(* IEC 61131-3 sources: JaccoSigma/tempclass/Class/SDM081, 1 file *)

(* ---- SDM081.st ---- *)
(*!
<Class
	Name               = "SDM081"
	Revision           = "1.11"
	RealtimeTask       = "false"
	CyclicTask         = "false"
	BackgroundTask     = "false"
	Sigmatek           = "true"
	OSInterface        = "false"
	HighPriority       = "false"
	Automatic          = "false"
	UpdateMode         = "Prescan"
	IconPath           = ".\Class\sdm.ico"
	SharedCommandTable = "true"
	Objectsize         = "(532,120)">
	<Channels>
		<Server Name="Safe_Input1" Visualized="true" Initialize="false" WriteProtected="true" Retentive="false" Comment="State of input (read only)&#13;&#10;&#13;&#10;-1..Error&#13;&#10; 0..Input Low&#13;&#10; 1..Input High"/>
		<Server Name="Safe_Input2" Visualized="true" Initialize="false" WriteProtected="true" Retentive="false" Comment="State of input (read only)&#13;&#10;&#13;&#10;-1..Error&#13;&#10; 0..Input Low&#13;&#10; 1..Input High"/>
		<Server Name="Safe_Input3" Visualized="true" Initialize="false" WriteProtected="true" Retentive="false" Comment="State of input (read only)&#13;&#10;&#13;&#10;-1..Error&#13;&#10; 0..Input Low&#13;&#10; 1..Input High"/>
		<Server Name="Safe_Input4" Visualized="true" Initialize="false" WriteProtected="true" Retentive="false" Comment="State of input (read only)&#13;&#10;&#13;&#10;-1..Error&#13;&#10; 0..Input Low&#13;&#10; 1..Input High"/>
		<Server Name="Safe_Input5" Visualized="true" Initialize="false" WriteProtected="true" Retentive="false" Comment="State of input (read only)&#13;&#10;&#13;&#10;-1..Error&#13;&#10; 0..Input Low&#13;&#10; 1..Input High"/>
		<Server Name="Safe_Input6" Visualized="true" Initialize="false" WriteProtected="true" Retentive="false" Comment="State of input (read only)&#13;&#10;&#13;&#10;-1..Error&#13;&#10; 0..Input Low&#13;&#10; 1..Input High"/>
		<Server Name="Safe_Output1" Visualized="true" Initialize="false" WriteProtected="true" Retentive="false" Comment="State of output (read only)&#13;&#10;&#13;&#10;-1..Error&#13;&#10; 0..Output Low&#13;&#10; 1..Output High"/>
		<Server Name="Safe_Output2" Visualized="true" Initialize="false" WriteProtected="true" Retentive="false" Comment="State of output (read only)&#13;&#10;&#13;&#10;-1..Error&#13;&#10; 0..Output Low&#13;&#10; 1..Output High"/>
		<Server Name="SafeIOError" Visualized="true" Initialize="false" WriteProtected="true" Retentive="false" Comment="Shows which safe in/outputs are in error.&#13;&#10;The in/outputs are bitcoded.&#13;&#10;Bit0 = Input1&#13;&#10;Bit1 = Input2&#13;&#10;Bit2 = Input3&#13;&#10;Bit3 = Input1&#13;&#10;Bit4 = Input2&#13;&#10;Bit5 = Input3&#13;&#10;Bit6 = Output1&#13;&#10;Bit7 = Output2"/>
		<Server Name="Unsafe_Output1" Visualized="true" Initialize="false" WriteProtected="false" Retentive="false" Comment="State of output (write only; default value: 0)&#13;&#10;&#13;&#10;If safety is given (output would be 1), you can still switch to zero by writing 0 to this server"/>
		<Server Name="Unsafe_Output2" Visualized="true" Initialize="false" WriteProtected="false" Retentive="false" Comment="State of output (write only; default value: 0)&#13;&#10;&#13;&#10;If safety is given (output would be 1), you can still switch to zero by writing 0 to this server"/>
	</Channels>
	<RevDoku>
		<Owner Company="Sigmatek" Author="EisMic"/>
		<Dokumentation Revision="1.11" Date="12.08.2019" Author="LazJos" Company="Sigmatek" Description="Added support for HWAlarms."/>
		<Dokumentation Revision="1.10" Date="08.06.2018" Author="RamAnd" Company="Sigmatek" Description="LASAL Hardware Description (.lhd) file has been updated."/>
		<Dokumentation Revision="1.9" Date="24.04.2018" Author="RamAnd" Company="Sigmatek" Description="Added server to show hardware version if this feature is supported by the safety firmware of the SCP."/>
		<Dokumentation Revision="1.8" Date="30.11.2017" Author="FurDom" Company="Sigmatek" Description="Added QuitComError server description to .lhd file"/>
		<Dokumentation Revision="1.7" Date="24.10.2016" Author="ZoePat" Company="Sigmatek" Description="Set the base class to visualized, so the embedded string object &quot;SerialNoStr&quot; can be used in the LSE."/>
		<Dokumentation Revision="1.6" Date="12.07.2016" Author="SeiChr" Company="Sigmatek" Description="Added Values for the total Current calculation. SA 31571"/>
		<Dokumentation Revision="1.5" Date="21.01.2016" Author="EisMic" Company="Sigmatek" Description="Outputs are now written in RtPostScan instead of RtPreScan to improve the reaction speed."/>
		<Dokumentation Revision="1.4" Date="16.04.2015" Author="EisMic" Company="Sigmatek" Description="Added support for graphical hardware editor."/>
		<Dokumentation Revision="1.3" Date="05.12.2014" Author="ZoePat" Company="Sigmatek" Description="The Status of the Output2 is now shown correctly at the Server."/>
		<Dokumentation Revision="1.2" Date="31.10.2014" Author="lanste" Company="Sigmatek" Description="Fixed error: Safe IO were displayed on wrong safety hardwareclass if the class is not required and not online.&#13;&#10;Fixed error: Safe IO were displayed on wrong safety hardwareclass if the hardware configuration did not match the project configuration.&#13;&#10;Set IOs to -2 if Class is not online."/>
		<Dokumentation Revision="1.1" Date="31.07.2014" Author="PieSte" Company="Sigmatek" Description="Added QuitComError server to quit errors on safety cpu."/>
		<Dokumentation Revision="1.0" Date="24.03.2013" Author="EisMic" Company="Sigmatek" Description="First library version"/>
	</RevDoku>
	<Network Name="SDM081">
		<!-- List of Components in this network -->
		<Components>
			<Object
				Name       = "_base"
				Class      = "SdiasSafetyBase"
				Position   = "(218,120)"
				Visualized = "true">
				<Channels>
					<Server Name="CallCommand"/>
					<Server Name="ClassState"/>
					<Server Name="DeviceID"/>
					<Server Name="HwVersion"/>
					<Server Name="QuitComError"/>
					<Server Name="RetryCounteruC1"/>
					<Server Name="RetryCounteruC2"/>
					<Server Name="SafetyNumber"/>
					<Server Name="SerialNo"/>
					<Client Name="InputsNeeded" Value="6"/>
					<Client Name="OutputsNeeded" Value="2"/>
					<Client Name="Place"/>
					<Client Name="Required" Value="1"/>
					<Client Name="SdiasSafetyIn"/>
					<Client Name="SetDeviceID" Value="2#101001"/>
				</Channels>
			</Object>
		</Components>
		<Comments>
		</Comments>
		<!-- List of Connections in this network -->
		<Connections>
			<Connection Source="this.ClassState" Destination="_base.ClassState" Vertices="(992,210),(820,210),"/>
			<Connection Source="_base.SdiasSafetyIn" Destination="this.SdiasSafetyIn" Vertices="(218,210),(38,210),"/>
			<Connection Source="_base.Place" Destination="this.Place" Vertices="(218,270),(38,270),"/>
			<Connection Source="this.DeviceID" Destination="_base.DeviceID" Vertices="(992,270),(820,270),"/>
			<Connection Source="_base.Required" Destination="this.Required" Vertices="(218,330),(38,330),"/>
			<Connection Source="this.SerialNo" Destination="_base.SerialNo" Vertices="(992,390),(820,390),"/>
			<Connection Source="this.SafetyNumber" Destination="_base.SafetyNumber" Vertices="(992,450),(820,450),"/>
			<Connection Source="this.RetryCounteruC1" Destination="_base.RetryCounteruC1" Vertices="(992,510),(820,510),"/>
			<Connection Source="this.RetryCounteruC2" Destination="_base.RetryCounteruC2" Vertices="(992,570),(820,570),"/>
			<Connection Source="this.QuitComError" Destination="_base.QuitComError" Vertices="(992,630),(820,690),"/>
			<Connection Source="this.HwVersion" Destination="_base.HwVersion" Vertices="(992,330),(820,330),"/>
		</Connections>
		<!-- Headerfiles -->
		<Options>
		</Options>
	</Network>
</Class>
*)
#pragma using SdiasSafetyBase

SDM081 : CLASS
: SdiasSafetyBase
  //Servers:
	Safe_Input1 	: SvrCh_DINT;
	Safe_Input2 	: SvrCh_DINT;
	Safe_Input3 	: SvrCh_DINT;
	Safe_Input4 	: SvrCh_DINT;
	Safe_Input5 	: SvrCh_DINT;
	Safe_Input6 	: SvrCh_DINT;
	Safe_Output1 	: SvrCh_DINT;
	Unsafe_Output1 	: SvrCh_DINT;
	Safe_Output2 	: SvrCh_DINT;
	Unsafe_Output2 	: SvrCh_DINT;
	SafeIOError 	: SvrCh_BDINT;
  //Clients:
  //Variables:
		TempInputState : ARRAY [0..9] OF DINT;

		Filter : ARRAY [0..9] OF DINT;

  //Functions:

	FUNCTION VIRTUAL GLOBAL Init;

	FUNCTION VIRTUAL GLOBAL RtWork
		VAR_INPUT
			EAX 	: UDINT;
		END_VAR
		VAR_OUTPUT
			state (EAX) 	: UDINT;
		END_VAR;
				//! <Function Comment="Called when class state was set to _NoHardware &#13;&#10;No Implementation Overload in derived classes if needed " Name="SetClassStateError"/>
	FUNCTION VIRTUAL SetClassStateError;

	FUNCTION VIRTUAL GLOBAL Unsafe_Output1::Write
		VAR_INPUT
			input (EAX) 	: DINT;
		END_VAR
		VAR_OUTPUT
			result (EAX) 	: DINT;
		END_VAR;

	FUNCTION VIRTUAL GLOBAL Unsafe_Output2::Write
		VAR_INPUT
			input (EAX) 	: DINT;
		END_VAR
		VAR_OUTPUT
			result (EAX) 	: DINT;
		END_VAR;
  //Tables:
	FUNCTION @STD
		VAR_OUTPUT
			ret_code	: CONFSTATES;
		END_VAR;
	FUNCTION GLOBAL TAB @CT_;
END_CLASS;

FUNCTION VIRTUAL GLOBAL SDM081::RtWork
	VAR_INPUT
		EAX 	: UDINT;
	END_VAR
	VAR_OUTPUT
		state (EAX) 	: UDINT;
	END_VAR

  // 0 = inputs, 1 = outputs
  if EAX = 0 then

#ifdef SB_SAFETY_INPUT_FILTER
    // if AcceptState bit is set => accept state
    if IOStates AND 2#10 then
      TempInputState[0] := to_dint(IOStates AND 2#1);

      if TempInputState[0] < Safe_Input1 then
        if Filter[0] <= 0 then
          Safe_Input1 := TempInputState[0];
        else
          Filter[0] -= 1;
        end_if;
      else
        Safe_Input1 := TempInputState[0];
        Filter[0] := SB_SAFETY_INPUT_FILTER;
      end_if;

      // show error state of this IO
      SafeIOError.1 := FALSE;
    else
      // otherwise, there's an error
      Safe_Input1 := -1;

      // show error state of this IO
      SafeIOError.1 := TRUE;
    end_if;

    // if AcceptState bit is set => accept state
    if IOStates AND 2#1000 then
      TempInputState[1] := to_dint(IOStates AND 2#100) SHR 2;

      if TempInputState[1] < Safe_Input2 then
        if Filter[1] <= 0 then
          Safe_Input2 := TempInputState[1];
        else
          Filter[1] -= 1;
        end_if;
      else
        Safe_Input2 := TempInputState[1];
        Filter[1] := SB_SAFETY_INPUT_FILTER;
      end_if;

      // show error state of this IO
      SafeIOError.2 := FALSE;
    else
      // otherwise, there's an error
      Safe_Input2 := -1;

      // show error state of this IO
      SafeIOError.2 := TRUE;
    end_if;

    // if AcceptState bit is set => accept state
    if IOStates AND 2#100000 then
      TempInputState[2] := to_dint(IOStates AND 2#10000) SHR 4;

      if TempInputState[2] < Safe_Input3 then
        if Filter[2] <= 0 then
          Safe_Input3 := TempInputState[2];
        else
          Filter[2] -= 1;
        end_if;
      else
        Safe_Input3 := TempInputState[2];
        Filter[2] := SB_SAFETY_INPUT_FILTER;
      end_if;

      // show error state of this IO
      SafeIOError.3 := FALSE;
    else
      // otherwise, there's an error
      Safe_Input3 := -1;

      // show error state of this IO
      SafeIOError.3 := TRUE;
    end_if;

    // if AcceptState bit is set => accept state
    if IOStates AND 2#10000000 then
      TempInputState[3] := to_dint(IOStates AND 2#1000000) SHR 6;

      if TempInputState[3] < Safe_Input4 then
        if Filter[3] <= 0 then
          Safe_Input4 := TempInputState[3];
        else
          Filter[3] -= 1;
        end_if;
      else
        Safe_Input4 := TempInputState[3];
        Filter[3] := SB_SAFETY_INPUT_FILTER;
      end_if;

      // show error state of this IO
      SafeIOError.4 := FALSE;
    else
      // otherwise, there's an error
      Safe_Input4 := -1;

      // show error state of this IO
      SafeIOError.4 := TRUE;
    end_if;

    // if AcceptState bit is set => accept state
    if IOStates AND 2#1000000000 then
      TempInputState[4] := to_dint(IOStates AND 2#100000000) SHR 8;

      if TempInputState[4] < Safe_Input5 then
        if Filter[4] <= 0 then
          Safe_Input5 := TempInputState[4];
        else
          Filter[4] -= 1;
        end_if;
      else
        Safe_Input5 := TempInputState[4];
        Filter[4] := SB_SAFETY_INPUT_FILTER;
      end_if;

      // show error state of this IO
      SafeIOError.5 := FALSE;
    else
      // otherwise, there's an error
      Safe_Input5 := -1;

      // show error state of this IO
      SafeIOError.5 := TRUE;
    end_if;

    // if AcceptState bit is set => accept state
    if IOStates AND 2#100000000000 then
      TempInputState[5] := to_dint(IOStates AND 2#10000000000) SHR 10;

      if TempInputState[5] < Safe_Input6 then
        if Filter[5] <= 0 then
          Safe_Input6 := TempInputState[5];
        else
          Filter[5] -= 1;
        end_if;
      else
        Safe_Input6 := TempInputState[5];
        Filter[5] := SB_SAFETY_INPUT_FILTER;
      end_if;

      // show error state of this IO
      SafeIOError.6 := FALSE;
    else
      // otherwise, there's an error
      Safe_Input6 := -1;

      // show error state of this IO
      SafeIOError.6 := TRUE;
    end_if;

#else

    // if AcceptState bit is set => accept state
    if IOStates AND 2#10 then
      Safe_Input1 := to_dint(IOStates AND 2#1);

      // show error state of this IO
      SafeIOError.1 := FALSE;
    else
      // otherwise, there's an error
      Safe_Input1 := -1;

      // show error state of this IO
      SafeIOError.1 := TRUE;
    end_if;

    // if AcceptState bit is set => accept state
    if IOStates AND 2#1000 then
      Safe_Input2 := to_dint(IOStates AND 2#100) SHR 2;

      // show error state of this IO
      SafeIOError.2 := FALSE;
    else
      // otherwise, there's an error
      Safe_Input2 := -1;

      // show error state of this IO
      SafeIOError.2 := TRUE;
    end_if;

    // if AcceptState bit is set => accept state
    if IOStates AND 2#100000 then
      Safe_Input3 := to_dint(IOStates AND 2#10000) SHR 4;

      // show error state of this IO
      SafeIOError.3 := FALSE;
    else
      // otherwise, there's an error
      Safe_Input3 := -1;

      // show error state of this IO
      SafeIOError.3 := TRUE;
    end_if;

    // if AcceptState bit is set => accept state
    if IOStates AND 2#10000000 then
      Safe_Input4 := to_dint(IOStates AND 2#1000000) SHR 6;

      // show error state of this IO
      SafeIOError.4 := FALSE;
    else
      // otherwise, there's an error
      Safe_Input4 := -1;

      // show error state of this IO
      SafeIOError.4 := TRUE;
    end_if;

    // if AcceptState bit is set => accept state
    if IOStates AND 2#1000000000 then
      Safe_Input5 := to_dint(IOStates AND 2#100000000) SHR 8;

      // show error state of this IO
      SafeIOError.5 := FALSE;
    else
      // otherwise, there's an error
      Safe_Input5 := -1;

      // show error state of this IO
      SafeIOError.5 := TRUE;
    end_if;

    // if AcceptState bit is set => accept state
    if IOStates AND 2#100000000000 then
      Safe_Input6 := to_dint(IOStates AND 2#10000000000) SHR 10;

      // show error state of this IO
      SafeIOError.6 := FALSE;
    else
      // otherwise, there's an error
      Safe_Input6 := -1;

      // show error state of this IO
      SafeIOError.6 := TRUE;
    end_if;
#endif

  //  EAX = 1 : Outputs
  else

  // if AcceptState bit is set => accept state
    if IOStates AND 2#10 then
      Safe_Output1 := to_dint(IOStates AND 2#1);

      // show error state of this IO
      SafeIOError.7 := FALSE;
    else
      // otherwise, there's an error
      Safe_Output1 := -1;

      // show error state of this IO
      SafeIOError.7 := TRUE;
    end_if;

    // if AcceptState bit is set => accept state
    if IOStates AND 2#1000 then
      Safe_Output2 := to_dint(IOStates AND 2#100) SHR 2;

      // show error state of this IO
      SafeIOError.8 := FALSE;
    else
      // otherwise, there's an error
      Safe_Output2 := -1;

      // show error state of this IO
      SafeIOError.8 := TRUE;
    end_if;

  end_if;

	state := READY;

END_FUNCTION

FUNCTION VIRTUAL GLOBAL SDM081::Unsafe_Output1::Write
	VAR_INPUT
		input (EAX) 	: DINT;
	END_VAR
	VAR_OUTPUT
		result (EAX) 	: DINT;
	END_VAR

  if input then
    result := Unsafe_Output1 := 1;
    UnsafeOutputStates.1 := TRUE;
  else
    result := Unsafe_Output1 := 0;
    UnsafeOutputStates.1 := FALSE;
  end_if;

END_FUNCTION

FUNCTION VIRTUAL GLOBAL SDM081::Unsafe_Output2::Write
	VAR_INPUT
		input (EAX) 	: DINT;
	END_VAR
	VAR_OUTPUT
		result (EAX) 	: DINT;
	END_VAR

  if input then
    result := Unsafe_Output2 := 1;
    UnsafeOutputStates.2 := TRUE;
  else
    result := Unsafe_Output2 := 0;
    UnsafeOutputStates.2 := FALSE;
  end_if;

END_FUNCTION

FUNCTION VIRTUAL GLOBAL SDM081::Init

  SdiasSafetyBase::Init();

  if us_FirstScan = 1 then
    Unsafe_Output1 := Unsafe_Output1 <> 0;
    Unsafe_Output2 := Unsafe_Output2 <> 0;

    UnsafeOutputStates.1 := to_bool(Unsafe_Output1);
    UnsafeOutputStates.2 := to_bool(Unsafe_Output2);

  end_if;

END_FUNCTION

FUNCTION VIRTUAL SDM081::SetClassStateError
  VAR
    i : UDINT;
    pServer : ^DINT;
  END_VAR

  pServer := #Safe_Input1;

  for i := 0 to 5 do
    pServer^ := SDIAS_SAFETY_INVALID_IO_NOHW;
    pServer += sizeof(SvrCh);
  end_for;

  Safe_Output1 := SDIAS_SAFETY_INVALID_IO_NOHW;
  Safe_Output2 := SDIAS_SAFETY_INVALID_IO_NOHW;

END_FUNCTION
